// TIA Portal V20 export
TYPE "typeCmInterfaceBrakeTest"
// stored: Access Published, Namespace Unit1.Em7
   STRUCT
      ngKicker : "LER_typeBrakeTestEmInterface";
      passKicker : "LER_typeBrakeTestEmInterface";
   END_STRUCT;
END_TYPE
